# EPICS substitutions: VCSIOCS/BSVIOC/bsviocApp/Db/userHost.substitutions
# Example substitutions file

file "db/dbExample1.db" {
    { user = "vcsHost" }
}

file db/dbExample2.db {
    pattern { user, no, scan }
        { "vcsHost", 1, "1 second" }
        { "vcsHost", 2, "2 second" }
        { "vcsHost", 3, "5 second" }
}
